(* CODESYS project xlh_rover_signal_test_00_01.project
   Description: Receives some incoming messages and echoes them with CAN-ID +1
   Company: 3S - Smart Software Solutions GmbH
   Version: 1.0.0.0
   Title: CAN Bus API Example
   Author: 3S - Smart Software Solutions GmbH

Project tree, tasks and I/O mapping:
  xLH_base : CODESYS Control for Raspberry Pi 64 SL, CODESYS, order no. 2302000009, version 4.18.0.0
    application app
      libraries: Standard, 3.5.18.0 (System); Util, 3.5.21.0 (System); VisuDialogs, * (System); Memory, * (3S - Smart Software Solutions GmbH); CmpBitmapPool, * (System); CAN API, 1.0.0.4 (CODESYS); MemoryUtils, * (3S - Smart Software Solutions GmbH); CAA CiA 405, 4.3.0.0 (CODESYS)
      task VISU_TASK (cyclic, interval 100 ms, priority 31) calls VisuElems.Visu_Prg
      task MAIN_TASK (cyclic, interval 10 ms, priority 1) calls MAIN_CALLER
      task ENIPAdapterIOTask (cyclic, interval t#1ms, priority 1) calls EtherNet_IP_Adapter.IOCycle
      task ENIPAdapterServiceTask (cyclic, interval t#20ms, priority 30) calls EtherNet_IP_Adapter.ServiceCycle
      program MAIN [ST]
      visualisation Visualization
      program MAIN_CALLER [ST]
      trace Trace (task MAIN_TASK): MAIN.diPosition, MAIN.auiUltrasonic[1], MAIN.iSpeedRight, MAIN.iSpeedLeft, MAIN.iPitch
    SoftMotion General Axis Pool
      a_axis : SM_Drive_PosControl, CODESYS, order no. 1805, version 4.18.0.0
          settings: wDriveID = 4; dwRatioTechUnitsDenom = 101846; iRatioTechUnitsNum = -125; eRampType = 1; fSWMaxVelocity = 50; fSWMaxAcceleration = 100; fSWMaxDeceleration = 100; fSWMaxJerk = 1000; fSWLimitNegative = -1000.0; ScalingIncs = 814768; ScalingUnits = 1000; InvertDirection = TRUE; IsLinearMotor = TRUE; MaximumOutputVelocityInt = 40738; MinimumOutputVelocityInt = -40738; Kp = 0.05; MaxFollowingError = 5.0; EnableFollowingErrorCheck = TRUE; DeadTime = 3.0
      x_axis : SM_Drive_PosControl, CODESYS, order no. 1805, version 4.18.0.0
          settings: dwRatioTechUnitsDenom = 101846; iRatioTechUnitsNum = 125; eRampType = 1; fSWMaxVelocity = 50; fSWMaxAcceleration = 100; fSWMaxDeceleration = 100; fSWMaxJerk = 1000; fSWLimitNegative = -1000; ScalingIncs = 814768; ScalingUnits = 1000; IsLinearMotor = TRUE; MaximumOutputVelocityInt = 40738; MinimumOutputVelocityInt = -40738; Kp = 0.05; MaxFollowingError = 5.0; EnableFollowingErrorCheck = TRUE; DeadTime = 3.0
      y_axis : SM_Drive_PosControl, CODESYS, order no. 1805, version 4.18.0.0
          settings: wDriveID = 2; dwRatioTechUnitsDenom = 101846; iRatioTechUnitsNum = 125; eRampType = 1; fSWMaxVelocity = 50; fSWMaxAcceleration = 100; fSWMaxDeceleration = 100; fSWMaxJerk = 1000; fSWLimitNegative = -1000; ScalingIncs = 814768; ScalingUnits = 1000; IsLinearMotor = TRUE; MaximumOutputVelocityInt = 40738; MinimumOutputVelocityInt = -40738; Kp = 0.05; MaxFollowingError = 5.0; EnableFollowingErrorCheck = TRUE; DeadTime = 3.0
      z_axis : SM_Drive_PosControl, CODESYS, order no. 1805, version 4.18.0.0
          settings: wDriveID = 3; dwRatioTechUnitsDenom = 101846; iRatioTechUnitsNum = 125; eRampType = 1; fSWMaxVelocity = 50; fSWMaxAcceleration = 100; fSWMaxDeceleration = 100; fSWMaxJerk = 1000; fSWLimitNegative = -1000; ScalingIncs = 814768; ScalingUnits = 1000; IsLinearMotor = TRUE; MaximumOutputVelocityInt = 40738; MinimumOutputVelocityInt = -40738; Kp = 0.05; MaxFollowingError = 5.0; EnableFollowingErrorCheck = TRUE; DeadTime = 3.0
    GPIOs_A_B : GPIOs B+/Pi2, CODESYS, version 4.15.0.0
        unmapped channels: digital inputs (GPIO0..GPIO31), digital outputs (GPIO0..GPIO31)
    Onewire
    Camera device
      <Leer>
    SPI
    I²C
    CANbus : CANbus, CODESYS, version 4.3.0.0
        settings: Baudrate = 1000 kbit/s
      CANopen_Manager : CANopen_Manager, CODESYS, version 4.3.0.0
          settings: ConfigVersion = 50659584
        xlh_ddsm210_ultrasonic : xlh_ddsm210_ultrasonic, xemax ag, order no. 0, version Revision=16#00000001, FileVersion=1.0
            settings: NODEIDSAVED = 1; SDO Timeout = 1000000; PDO_Autoconfig = FALSE; EXPERTSETTINGS = FALSE; Sync-General Parameters.Sync-COBID = 16#00000080; Sync-General Parameters.Communication Cycle Period = 16#00000000 usec; PDO 16#1400.COBID = 16#00000201; Process by CANopenManager = TRUE; PDO 16#1800.COBID = 16#00000181; Process by CANopenManager = TRUE; PDO 16#1801.COBID = 16#00000281; Process by CANopenManager = TRUE; PDO 16#1802.COBID = 16#00000381; Process by CANopenManager = TRUE; PDO 16#1803.COBID = 16#00000481; Process by CANopenManager = TRUE; set_speed.Subindex = 16#01; set_current_limit.Subindex = 16#01; set_acc_time.Subindex = 16#01; set_cmd.Subindex = 16#01; speed.Subindex = 16#01; current.Subindex = 16#01; acc_time.Subindex = 16#01; temperature.Subindex = 16#01; position.Subindex = 16#01; error_code.Subindex = 16#01; ultrasonic_1.Subindex = 16#01; ultrasonic_2.Subindex = 16#02; ultrasonic_3.Subindex = 16#03; debug_1.Subindex = 16#02; ultrasonic_4.Subindex = 16#04; ultrasonic_5.Subindex = 16#05; ultrasonic_6.Subindex = 16#06; debug_2.Subindex = 16#03; SDO List.Set COB-ID sync.Index = 16#1005; SDO List.Set COB-ID sync.Subindex = 16#00; SDO List.Set COB-ID sync.Value = 16#00000080; SDO List.Set COB-ID sync.Size = 32; SDO List.Set COB-ID sync.AbortIfError = FALSE; SDO List.Set COB-ID sync.JumpToLine = FALSE;
              SDO List.Set COB-ID sync.Line = 0; SDO List.Set communication cycle period.Index = 16#1006; SDO List.Set communication cycle period.Subindex = 16#00; SDO List.Set communication cycle period.Value = 16#00000000; SDO List.Set communication cycle period.Size = 32; SDO List.Set communication cycle period.AbortIfError = FALSE; SDO List.Set communication cycle period.JumpToLine = FALSE; SDO List.Set communication cycle period.Line = 0; SDO List.Set Guardtime.Index = 16#100C; SDO List.Set Guardtime.Subindex = 16#00; SDO List.Set Guardtime.Value = 16#000000C8; SDO List.Set Guardtime.Size = 16; SDO List.Set Guardtime.AbortIfError = FALSE; SDO List.Set Guardtime.JumpToLine = FALSE; SDO List.Set Guardtime.Line = 0; SDO List.Set Lifetime.Index = 16#100D; SDO List.Set Lifetime.Subindex = 16#00; SDO List.Set Lifetime.Value = 16#00000003; SDO List.Set Lifetime.Size = 8; SDO List.Set Lifetime.AbortIfError = FALSE; SDO List.Set Lifetime.JumpToLine = FALSE; SDO List.Set Lifetime.Line = 0; SDO List.Set Heartbeat Consumer.Index = 16#1016; SDO List.Set Heartbeat Consumer.Subindex = 16#01; SDO List.Set Heartbeat Consumer.Value = 0; SDO List.Set Heartbeat Consumer.Size = 32; SDO List.Set Heartbeat Consumer.AbortIfError = FALSE; SDO List.Set Heartbeat Consumer.JumpToLine = FALSE; SDO List.Set Heartbeat Consumer.Line = 0; SDO List.Disable PDO.Index = 16#1400; SDO List.Disable PDO.Subindex = 16#01; SDO List.Disable PDO.Value = 16#80000201; SDO List.Disable PDO.Size = 32; SDO List.Disable PDO.AbortIfError = FALSE; SDO List.Disable PDO.JumpToLine = FALSE; SDO List.Disable PDO.Line = 0; SDO List.Set transmission type.Index = 16#1400; SDO List.Set transmission type.Subindex = 16#02; SDO List.Set transmission type.Value = 16#FF; SDO List.Set transmission type.Size = 8;
              SDO List.Set transmission type.AbortIfError = FALSE; SDO List.Set transmission type.JumpToLine = FALSE; SDO List.Set transmission type.Line = 0; SDO List.Set and enable COB-ID.Index = 16#1400; SDO List.Set and enable COB-ID.Subindex = 16#01; SDO List.Set and enable COB-ID.Value = 16#00000201; SDO List.Set and enable COB-ID.Size = 32; SDO List.Set and enable COB-ID.AbortIfError = FALSE; SDO List.Set and enable COB-ID.JumpToLine = FALSE; SDO List.Set and enable COB-ID.Line = 0; SDO List.Disable PDO.Index = 16#1800; SDO List.Disable PDO.Subindex = 16#01; SDO List.Disable PDO.Value = 16#80000181; SDO List.Disable PDO.Size = 32; SDO List.Disable PDO.AbortIfError = FALSE; SDO List.Disable PDO.JumpToLine = FALSE; SDO List.Disable PDO.Line = 0; SDO List.Set transmission type.Index = 16#1800; SDO List.Set transmission type.Subindex = 16#02; SDO List.Set transmission type.Value = 16#FF; SDO List.Set transmission type.Size = 8; SDO List.Set transmission type.AbortIfError = FALSE; SDO List.Set transmission type.JumpToLine = FALSE; SDO List.Set transmission type.Line = 0; SDO List.Set inhibit time.Index = 16#1800; SDO List.Set inhibit time.Subindex = 16#03; SDO List.Set inhibit time.Value = 16#0000; SDO List.Set inhibit time.Size = 16; SDO List.Set inhibit time.AbortIfError = FALSE; SDO List.Set inhibit time.JumpToLine = FALSE; SDO List.Set inhibit time.Line = 0; SDO List.Set event time.Index = 16#1800; SDO List.Set event time.Subindex = 16#05; SDO List.Set event time.Value = 16#0000; SDO List.Set event time.Size = 16; SDO List.Set event time.AbortIfError = FALSE; SDO List.Set event time.JumpToLine = FALSE; SDO List.Set event time.Line = 0; SDO List.Set and enable COB-ID.Index = 16#1800; SDO List.Set and enable COB-ID.Subindex = 16#01;
              SDO List.Set and enable COB-ID.Value = 16#00000181; SDO List.Set and enable COB-ID.Size = 32; SDO List.Set and enable COB-ID.AbortIfError = FALSE; SDO List.Set and enable COB-ID.JumpToLine = FALSE; SDO List.Set and enable COB-ID.Line = 0; SDO List.Disable PDO.Index = 16#1801; SDO List.Disable PDO.Subindex = 16#01; SDO List.Disable PDO.Value = 16#80000281; SDO List.Disable PDO.Size = 32; SDO List.Disable PDO.AbortIfError = FALSE; SDO List.Disable PDO.JumpToLine = FALSE; SDO List.Disable PDO.Line = 0; SDO List.Set transmission type.Index = 16#1801; SDO List.Set transmission type.Subindex = 16#02; SDO List.Set transmission type.Value = 16#FF; SDO List.Set transmission type.Size = 8; SDO List.Set transmission type.AbortIfError = FALSE; SDO List.Set transmission type.JumpToLine = FALSE; SDO List.Set transmission type.Line = 0; SDO List.Set inhibit time.Index = 16#1801; SDO List.Set inhibit time.Subindex = 16#03; SDO List.Set inhibit time.Value = 16#0000; SDO List.Set inhibit time.Size = 16; SDO List.Set inhibit time.AbortIfError = FALSE; SDO List.Set inhibit time.JumpToLine = FALSE; SDO List.Set inhibit time.Line = 0; SDO List.Set event time.Index = 16#1801; SDO List.Set event time.Subindex = 16#05; SDO List.Set event time.Value = 16#0000; SDO List.Set event time.Size = 16; SDO List.Set event time.AbortIfError = FALSE; SDO List.Set event time.JumpToLine = FALSE; SDO List.Set event time.Line = 0; SDO List.Set and enable COB-ID.Index = 16#1801; SDO List.Set and enable COB-ID.Subindex = 16#01; SDO List.Set and enable COB-ID.Value = 16#00000281; SDO List.Set and enable COB-ID.Size = 32; SDO List.Set and enable COB-ID.AbortIfError = FALSE; SDO List.Set and enable COB-ID.JumpToLine = FALSE; SDO List.Set and enable COB-ID.Line = 0;
              SDO List.Disable PDO.Index = 16#1802; SDO List.Disable PDO.Subindex = 16#01; SDO List.Disable PDO.Value = 16#80000381; SDO List.Disable PDO.Size = 32; SDO List.Disable PDO.AbortIfError = FALSE; SDO List.Disable PDO.JumpToLine = FALSE; SDO List.Disable PDO.Line = 0; SDO List.Set transmission type.Index = 16#1802; SDO List.Set transmission type.Subindex = 16#02; SDO List.Set transmission type.Value = 16#FF; SDO List.Set transmission type.Size = 8; SDO List.Set transmission type.AbortIfError = FALSE; SDO List.Set transmission type.JumpToLine = FALSE; SDO List.Set transmission type.Line = 0; SDO List.Set inhibit time.Index = 16#1802; SDO List.Set inhibit time.Subindex = 16#03; SDO List.Set inhibit time.Value = 16#0000; SDO List.Set inhibit time.Size = 16; SDO List.Set inhibit time.AbortIfError = FALSE; SDO List.Set inhibit time.JumpToLine = FALSE; SDO List.Set inhibit time.Line = 0; SDO List.Set event time.Index = 16#1802; SDO List.Set event time.Subindex = 16#05; SDO List.Set event time.Value = 16#0000; SDO List.Set event time.Size = 16; SDO List.Set event time.AbortIfError = FALSE; SDO List.Set event time.JumpToLine = FALSE; SDO List.Set event time.Line = 0; SDO List.Set and enable COB-ID.Index = 16#1802; SDO List.Set and enable COB-ID.Subindex = 16#01; SDO List.Set and enable COB-ID.Value = 16#00000381; SDO List.Set and enable COB-ID.Size = 32; SDO List.Set and enable COB-ID.AbortIfError = FALSE; SDO List.Set and enable COB-ID.JumpToLine = FALSE; SDO List.Set and enable COB-ID.Line = 0; SDO List.Disable PDO.Index = 16#1803; SDO List.Disable PDO.Subindex = 16#01; SDO List.Disable PDO.Value = 16#80000481; SDO List.Disable PDO.Size = 32; SDO List.Disable PDO.AbortIfError = FALSE;
              SDO List.Disable PDO.JumpToLine = FALSE; SDO List.Disable PDO.Line = 0; SDO List.Set transmission type.Index = 16#1803; SDO List.Set transmission type.Subindex = 16#02; SDO List.Set transmission type.Value = 16#FF; SDO List.Set transmission type.Size = 8; SDO List.Set transmission type.AbortIfError = FALSE; SDO List.Set transmission type.JumpToLine = FALSE; SDO List.Set transmission type.Line = 0; SDO List.Set inhibit time.Index = 16#1803; SDO List.Set inhibit time.Subindex = 16#03; SDO List.Set inhibit time.Value = 16#0000; SDO List.Set inhibit time.Size = 16; SDO List.Set inhibit time.AbortIfError = FALSE; SDO List.Set inhibit time.JumpToLine = FALSE; SDO List.Set inhibit time.Line = 0; SDO List.Set event time.Index = 16#1803; SDO List.Set event time.Subindex = 16#05; SDO List.Set event time.Value = 16#0000; SDO List.Set event time.Size = 16; SDO List.Set event time.AbortIfError = FALSE; SDO List.Set event time.JumpToLine = FALSE; SDO List.Set event time.Line = 0; SDO List.Set and enable COB-ID.Index = 16#1803; SDO List.Set and enable COB-ID.Subindex = 16#01; SDO List.Set and enable COB-ID.Value = 16#00000481; SDO List.Set and enable COB-ID.Size = 32; SDO List.Set and enable COB-ID.AbortIfError = FALSE; SDO List.Set and enable COB-ID.JumpToLine = FALSE; SDO List.Set and enable COB-ID.Line = 0; ConfigVersion = 50659584
            output app.MAIN.iSetSpeedLeft : INT  // set_speed
            output app.MAIN.iSetCurrentLimit : INT  // set_current_limit
            output app.MAIN.bySetAccTime : USINT  // set_acc_time
            output app.MAIN.bySetCmd : USINT  // set_cmd
            input  app.MAIN.iSpeedLeft : INT  // speed
            input  app.MAIN.iCurrentLeft : INT  // current
            input  app.MAIN.byAccTimeLeft : USINT  // acc_time
            input  app.MAIN.byTemperatureLeft : USINT  // temperature
            input  app.MAIN.diPositionLeft : DINT  // position
            input  app.MAIN.uiErrorCodeLeft : UINT  // error_code
            input  app.MAIN.uiUltrasonicRear : UINT  // ultrasonic_1
            input  app.MAIN.uiUltrasonicRearRight : UINT  // ultrasonic_2
            input  app.MAIN.uiUltrasonicFrontRight : UINT  // ultrasonic_3
            input  app.MAIN.uiUltrasonicFront : UINT  // ultrasonic_4
            input  app.MAIN.uiUltrasonicFrontLeft : UINT  // ultrasonic_5
            input  app.MAIN.uiUltrasonicRearLeft : UINT  // ultrasonic_6
            unmapped channels: debug_1, debug_2
        xlh_ddsm210_imu : xlh_ddsm210_imu, xemax ag, order no. 0, version Revision=16#00000001, FileVersion=1.0
            settings: NODEIDSAVED = 2; SDO Timeout = 1000000; EXPERTSETTINGS = FALSE; Sync-General Parameters.Sync-COBID = 16#00000080; Sync-General Parameters.Communication Cycle Period = 16#00000000 usec; PDO 16#1400.COBID = 16#00000202; Process by CANopenManager = TRUE; PDO 16#1800.COBID = 16#00000182; Process by CANopenManager = TRUE; PDO 16#1801.COBID = 16#00000282; Process by CANopenManager = TRUE; PDO 16#1802.COBID = 16#00000382; Process by CANopenManager = TRUE; set_speed.Subindex = 16#01; set_current_limit.Subindex = 16#01; set_acc_time.Subindex = 16#01; set_cmd.Subindex = 16#01; speed.Subindex = 16#01; current.Subindex = 16#01; acc_time.Subindex = 16#01; temperature.Subindex = 16#01; position.Subindex = 16#01; error_code.Subindex = 16#01; debug_1.Subindex = 16#02; yaw.Subindex = 16#01; pitch.Subindex = 16#02; roll.Subindex = 16#03; debug_2.Subindex = 16#03; SDO List.Set COB-ID sync.Index = 16#1005; SDO List.Set COB-ID sync.Subindex = 16#00; SDO List.Set COB-ID sync.Value = 16#00000080; SDO List.Set COB-ID sync.Size = 32; SDO List.Set COB-ID sync.AbortIfError = FALSE; SDO List.Set COB-ID sync.JumpToLine = FALSE; SDO List.Set COB-ID sync.Line = 0; SDO List.Set communication cycle period.Index = 16#1006; SDO List.Set communication cycle period.Subindex = 16#00; SDO List.Set communication cycle period.Value = 16#00000000; SDO List.Set communication cycle period.Size = 32; SDO List.Set communication cycle period.AbortIfError = FALSE;
              SDO List.Set communication cycle period.JumpToLine = FALSE; SDO List.Set communication cycle period.Line = 0; SDO List.Set Guardtime.Index = 16#100C; SDO List.Set Guardtime.Subindex = 16#00; SDO List.Set Guardtime.Value = 16#000000C8; SDO List.Set Guardtime.Size = 16; SDO List.Set Guardtime.AbortIfError = FALSE; SDO List.Set Guardtime.JumpToLine = FALSE; SDO List.Set Guardtime.Line = 0; SDO List.Set Lifetime.Index = 16#100D; SDO List.Set Lifetime.Subindex = 16#00; SDO List.Set Lifetime.Value = 16#00000003; SDO List.Set Lifetime.Size = 8; SDO List.Set Lifetime.AbortIfError = FALSE; SDO List.Set Lifetime.JumpToLine = FALSE; SDO List.Set Lifetime.Line = 0; SDO List.Set Heartbeat Consumer.Index = 16#1016; SDO List.Set Heartbeat Consumer.Subindex = 16#01; SDO List.Set Heartbeat Consumer.Value = 0; SDO List.Set Heartbeat Consumer.Size = 32; SDO List.Set Heartbeat Consumer.AbortIfError = FALSE; SDO List.Set Heartbeat Consumer.JumpToLine = FALSE; SDO List.Set Heartbeat Consumer.Line = 0; SDO List.Disable PDO.Index = 16#1400; SDO List.Disable PDO.Subindex = 16#01; SDO List.Disable PDO.Value = 16#80000202; SDO List.Disable PDO.Size = 32; SDO List.Disable PDO.AbortIfError = FALSE; SDO List.Disable PDO.JumpToLine = FALSE; SDO List.Disable PDO.Line = 0; SDO List.Set transmission type.Index = 16#1400; SDO List.Set transmission type.Subindex = 16#02; SDO List.Set transmission type.Value = 16#FF; SDO List.Set transmission type.Size = 8; SDO List.Set transmission type.AbortIfError = FALSE; SDO List.Set transmission type.JumpToLine = FALSE; SDO List.Set transmission type.Line = 0; SDO List.Set and enable COB-ID.Index = 16#1400; SDO List.Set and enable COB-ID.Subindex = 16#01; SDO List.Set and enable COB-ID.Value = 16#00000202;
              SDO List.Set and enable COB-ID.Size = 32; SDO List.Set and enable COB-ID.AbortIfError = FALSE; SDO List.Set and enable COB-ID.JumpToLine = FALSE; SDO List.Set and enable COB-ID.Line = 0; SDO List.Disable PDO.Index = 16#1800; SDO List.Disable PDO.Subindex = 16#01; SDO List.Disable PDO.Value = 16#80000182; SDO List.Disable PDO.Size = 32; SDO List.Disable PDO.AbortIfError = FALSE; SDO List.Disable PDO.JumpToLine = FALSE; SDO List.Disable PDO.Line = 0; SDO List.Set transmission type.Index = 16#1800; SDO List.Set transmission type.Subindex = 16#02; SDO List.Set transmission type.Value = 16#FF; SDO List.Set transmission type.Size = 8; SDO List.Set transmission type.AbortIfError = FALSE; SDO List.Set transmission type.JumpToLine = FALSE; SDO List.Set transmission type.Line = 0; SDO List.Set inhibit time.Index = 16#1800; SDO List.Set inhibit time.Subindex = 16#03; SDO List.Set inhibit time.Value = 16#0000; SDO List.Set inhibit time.Size = 16; SDO List.Set inhibit time.AbortIfError = FALSE; SDO List.Set inhibit time.JumpToLine = FALSE; SDO List.Set inhibit time.Line = 0; SDO List.Set event time.Index = 16#1800; SDO List.Set event time.Subindex = 16#05; SDO List.Set event time.Value = 16#0000; SDO List.Set event time.Size = 16; SDO List.Set event time.AbortIfError = FALSE; SDO List.Set event time.JumpToLine = FALSE; SDO List.Set event time.Line = 0; SDO List.Set and enable COB-ID.Index = 16#1800; SDO List.Set and enable COB-ID.Subindex = 16#01; SDO List.Set and enable COB-ID.Value = 16#00000182; SDO List.Set and enable COB-ID.Size = 32; SDO List.Set and enable COB-ID.AbortIfError = FALSE; SDO List.Set and enable COB-ID.JumpToLine = FALSE; SDO List.Set and enable COB-ID.Line = 0; SDO List.Disable PDO.Index = 16#1801;
              SDO List.Disable PDO.Subindex = 16#01; SDO List.Disable PDO.Value = 16#80000282; SDO List.Disable PDO.Size = 32; SDO List.Disable PDO.AbortIfError = FALSE; SDO List.Disable PDO.JumpToLine = FALSE; SDO List.Disable PDO.Line = 0; SDO List.Set transmission type.Index = 16#1801; SDO List.Set transmission type.Subindex = 16#02; SDO List.Set transmission type.Value = 16#FF; SDO List.Set transmission type.Size = 8; SDO List.Set transmission type.AbortIfError = FALSE; SDO List.Set transmission type.JumpToLine = FALSE; SDO List.Set transmission type.Line = 0; SDO List.Set inhibit time.Index = 16#1801; SDO List.Set inhibit time.Subindex = 16#03; SDO List.Set inhibit time.Value = 16#0000; SDO List.Set inhibit time.Size = 16; SDO List.Set inhibit time.AbortIfError = FALSE; SDO List.Set inhibit time.JumpToLine = FALSE; SDO List.Set inhibit time.Line = 0; SDO List.Set event time.Index = 16#1801; SDO List.Set event time.Subindex = 16#05; SDO List.Set event time.Value = 16#0000; SDO List.Set event time.Size = 16; SDO List.Set event time.AbortIfError = FALSE; SDO List.Set event time.JumpToLine = FALSE; SDO List.Set event time.Line = 0; SDO List.Set and enable COB-ID.Index = 16#1801; SDO List.Set and enable COB-ID.Subindex = 16#01; SDO List.Set and enable COB-ID.Value = 16#00000282; SDO List.Set and enable COB-ID.Size = 32; SDO List.Set and enable COB-ID.AbortIfError = FALSE; SDO List.Set and enable COB-ID.JumpToLine = FALSE; SDO List.Set and enable COB-ID.Line = 0; SDO List.Disable PDO.Index = 16#1802; SDO List.Disable PDO.Subindex = 16#01; SDO List.Disable PDO.Value = 16#80000382; SDO List.Disable PDO.Size = 32; SDO List.Disable PDO.AbortIfError = FALSE; SDO List.Disable PDO.JumpToLine = FALSE;
              SDO List.Disable PDO.Line = 0; SDO List.Set transmission type.Index = 16#1802; SDO List.Set transmission type.Subindex = 16#02; SDO List.Set transmission type.Value = 16#FF; SDO List.Set transmission type.Size = 8; SDO List.Set transmission type.AbortIfError = FALSE; SDO List.Set transmission type.JumpToLine = FALSE; SDO List.Set transmission type.Line = 0; SDO List.Set inhibit time.Index = 16#1802; SDO List.Set inhibit time.Subindex = 16#03; SDO List.Set inhibit time.Value = 16#0000; SDO List.Set inhibit time.Size = 16; SDO List.Set inhibit time.AbortIfError = FALSE; SDO List.Set inhibit time.JumpToLine = FALSE; SDO List.Set inhibit time.Line = 0; SDO List.Set event time.Index = 16#1802; SDO List.Set event time.Subindex = 16#05; SDO List.Set event time.Value = 16#0000; SDO List.Set event time.Size = 16; SDO List.Set event time.AbortIfError = FALSE; SDO List.Set event time.JumpToLine = FALSE; SDO List.Set event time.Line = 0; SDO List.Set and enable COB-ID.Index = 16#1802; SDO List.Set and enable COB-ID.Subindex = 16#01; SDO List.Set and enable COB-ID.Value = 16#00000382; SDO List.Set and enable COB-ID.Size = 32; SDO List.Set and enable COB-ID.AbortIfError = FALSE; SDO List.Set and enable COB-ID.JumpToLine = FALSE; SDO List.Set and enable COB-ID.Line = 0; ConfigVersion = 50659584
            output app.MAIN.iSetSpeedRight : INT  // set_speed
            output app.MAIN.iSetCurrentLimit : INT  // set_current_limit
            output app.MAIN.bySetAccTime : USINT  // set_acc_time
            output app.MAIN.bySetCmd : USINT  // set_cmd
            input  app.MAIN.iSpeedRight : INT  // speed
            input  app.MAIN.iCurrentRight : INT  // current
            input  app.MAIN.byAccTimeRight : USINT  // acc_time
            input  app.MAIN.byTemperatureRight : USINT  // temperature
            input  app.MAIN.diPositionRight : DINT  // position
            input  app.MAIN.uiErrorCodeRight : UINT  // error_code
            input  app.MAIN.iYaw : INT  // yaw
            input  app.MAIN.iPitch : INT  // pitch
            input  app.MAIN.iRoll : INT  // roll
            unmapped channels: debug_1, debug_2
    Ethernet : Ethernet, CODESYS, version 4.2.0.0
        settings: IPAddress = [192,168,1,189]; SubnetMask = [255,255,255,0]; GatewayAddress = [192,168,1,1]; MACAddress = [16#00,16#00,16#00,16#00,16#00,16#00]; NetworkInterfaceName = 'wlan0'; NetworkInterfaceName = "wlan0"; SaveCommunicationSettings = FALSE; IPAddress = [192,168,0,2]; SubnetMask = [255,255,255,0]; GatewayAddress = [0,0,0,0]
      EtherNet_IP_Adapter : EtherNet/IP Adapter, CODESYS, version 4.8.0.0
          settings: DeviceInfo.ProductName = 'xlh_rover_signal_test'; DeviceInfo.ProductCode = 1101; DeviceInfo.MajorRevision = 2; Number of Assemblies = 5; Number of Connections = 3; Connection Settings.Connection Number = 0; Connection Settings.Trigger and Transport = 67305474; Connection Settings.Connection Parameters = 4284744709; Connection Settings.O->T Requested packet interval (µs) = 0; Connection Settings.O->T Size (Bytes) = 0; Connection Settings.T->O Requested packet interval (µs) = 0; Connection Settings.T->O Size (Bytes) = 0; Connection Settings.Target Config Size (Bytes) = 2; Connection Settings.Connection Path Size (Bytes) = 8; Connection Settings.Connection Number = 1; Connection Settings.Trigger and Transport = 33751042; Connection Settings.Connection Parameters = 4284744453; Connection Settings.O->T Requested packet interval (µs) = 0; Connection Settings.O->T Size (Bytes) = 0; Connection Settings.T->O Requested packet interval (µs) = 0; Connection Settings.T->O Size (Bytes) = 0; Connection Settings.Target Config Size (Bytes) = 0; Connection Settings.Connection Path Size (Bytes) = 6; Connection Settings.Connection Number = 2; Connection Settings.Trigger and Transport = 16973826; Connection Settings.Connection Parameters = 4284744453; Connection Settings.O->T Requested packet interval (µs) = 0; Connection Settings.O->T Size (Bytes) = 0; Connection Settings.T->O Requested packet interval (µs) = 0; Connection Settings.T->O Size (Bytes) = 0; Connection Settings.Target Config Size (Bytes) = 0; Connection Settings.Connection Path Size (Bytes) = 6; Connection Path = [16#20,16#04,16#24,16#66,16#2C,16#64,16#2C,16#65]; Connection Path = [16#20,16#04,16#2C,16#C6,16#2C,16#65]; Connection Path = [16#20,16#04,16#2C,16#C7,16#2C,16#65]; Default Connection Path = [16#20,16#04,16#24,16#66,16#2C,16#64,16#2C,16#65]; Default Connection Path = [16#20,16#04,16#2C,16#C6,16#2C,16#65]; Default Connection Path = [16#20,16#04,16#2C,16#C7,16#2C,16#65]
        EtherNet_IP_Module : EtherNet/IP Module, CODESYS, version 4.6.0.0
            settings: ConsumingAssemblyID = 100; ProducingAssemblyID = 101; fJoystickXnorm.ReadOnly = False; fJoystickXnorm.BitSize = 64; fJoystickXnorm.DataSize = 8; fJoystickYnorm.ReadOnly = False; fJoystickYnorm.BitSize = 64; fJoystickYnorm.DataSize = 8; bySwitch.ReadOnly = False; byButton.ReadOnly = False; byLedSwitch.ReadOnly = False; byLedButton.ReadOnly = False; ConfigVersion = 50663168
            input  app.MAIN.fJoystickXnorm : LREAL  // fJoystickXnorm
            input  app.MAIN.fJoystickYnorm : LREAL  // fJoystickYnorm
            input  app.MAIN.bySwitch : BYTE  // bySwitch
            input  app.MAIN.byButton : BYTE  // byButton
            output app.MAIN.byLedSwitch : BYTE  // byLedSwitch
            output app.MAIN.byLedButton : BYTE  // byLedButton
  libraries: VisuSymbols, 4.5.0.0 (System); DepictorBase, 1.2.0.0 (CODESYS)
  text list GlobalTextList
  5ce3da45-db07-42e7-a21c-a00fff4ed8f6|C:\Users\phe\Downloads\Musterloesung_FUP.PNG
*)

// xLH_base/app/MAIN_CALLER
PROGRAM MAIN_CALLER
VAR
	bDevicesCoRunning: BOOL;
	fbTonDevicesCoRunning: TON := (PT:=T#250MS);
END_VAR

// Ueberwachung ob alle CAN-Open Devices im Status RUN sind
fbTonDevicesCoRunning(IN:= 
	(xlh_ddsm210_ultrasonic.CANopenState = _3SCOS.DEVICE_STATE.OPERATIONAL) AND
	(xlh_ddsm210_imu.CANopenState = _3SCOS.DEVICE_STATE.OPERATIONAL)
);

// falls alle Devices im Status RUN sind (inklusive Verzögerung), wird die POE MAIN aufgerufen
IF fbTonDevicesCoRunning.Q THEN
	MAIN();
END_IF

END_PROGRAM

// xLH_base/app/MAIN
PROGRAM MAIN
VAR_INPUT
	iSpeedLeft: INT;
	iSpeedRight: INT;
	iCurrentLeft: INT;
	iCurrentRight: INT;
	byAccTimeLeft: BYTE;
	byAccTimeRight: BYTE;
	byTemperatureLeft: BYTE;
	byTemperatureRight: BYTE;
	diPositionLeft: DINT;// still errors in the calculation => set to zero in the fw
	diPositionRight: DINT;// still errors in the calculation => set to zero in the fw
	{attribute 'displaymode':='hex'} 
	uiErrorCodeLeft: UINT;
	uiErrorCodeRight: UINT;
	uiUltrasonicFront: UINT;
	uiUltrasonicFrontLeft: UINT;
	uiUltrasonicFrontRight: UINT;
	uiUltrasonicRear: UINT;
	uiUltrasonicRearLeft: UINT;
	uiUltrasonicRearRight: UINT;
	
	
	iYaw: INT;
	iPitch: INT;
	iRoll: INT;
	fYaw: LREAL;
	fPitch: LREAL;
	fRoll: LREAL;
	
	// Ethernet IP
	fJoystickXnorm: LREAL;
	fJoystickYnorm: LREAL;
	bySwitch: BYTE;
	byButton: BYTE;
	iDebugRead: INT;
END_VAR
VAR_OUTPUT
	iSetSpeedLeft: INT := 0;
	iSetSpeedRight: INT := 0;
	iSetCurrentLimit: INT := 1000;// deactivated in the fw
	bySetAccTime: BYTE := 5;
	bySetCmd: BYTE := 0;
	
	// Ethernet IP
	byLedSwitch: BYTE;
	byLedButton: BYTE;
	iDebugWrite: INT;
END_VAR
VAR
	fSetSpeedLeft: LREAL;
	fSetSpeedRight: LREAL;
	
	byDummy: BYTE;
	iDummy: INT;
	uiDummy: UINT;
	diDummy: DINT;
	udiDummy: UDINT;

	fbBlink: BLINK := (TIMEHIGH:=T#100MS, TIMELOW:=T#100MS, ENABLE:=TRUE);
	fDummy: LREAL;
	
	unpackByte: MEM.UnpackByte;	
	abSwitch: ARRAY [0..7] OF BOOL;
	abButton: ARRAY [0..7] OF BOOL;
END_VAR
VAR CONSTANT
	fSpeedMax: LREAL := 500.0;
	fSpeedMaxDir: LREAL := 250.0;
END_VAR

fSetSpeedLeft := fJoystickYnorm * fSpeedMax * (1.0) + ABS(MAX(fJoystickXnorm, 0.0)) * fSpeedMaxDir * (1.0);
fSetSpeedRight := fJoystickYnorm * fSpeedMax * (-1.0) + ABS(MIN(fJoystickXnorm, 0.0)) * fSpeedMaxDir * (-1.0);

iSetSpeedLeft := TO_INT(fSetSpeedLeft);
iSetSpeedRight := TO_INT(fSetSpeedRight);
byDummy := bySetAccTime;

iDummy := iSpeedLeft;// -2100 ~ 2100 -> -210 ~ 210 rpm
iDummy := iSpeedRight;// -2100 ~ 2100 -> -210 ~ 210 rpm
iDummy := iCurrentLeft;// mA
iDummy := iCurrentRight;// mA
byDummy := byAccTimeLeft;// When it is set to 1, the acceleration time per 1rpm is 0.1ms. When it is set to 10, the acceleration time per 1rpm is 10*0.1 ms=1ms.
byDummy := byTemperatureLeft;// °C
uiDummy := uiUltrasonicFront;// resolution 0.1mm => 1000 ~ 100.0mm
uiDummy := uiUltrasonicFrontRight;// resolution 0.1mm => 1000 ~ 100.0mm
uiDummy := uiUltrasonicFrontLeft;// resolution 0.1mm => 1000 ~ 100.0mm
uiDummy := uiUltrasonicRear;// resolution 0.1mm => 1000 ~ 100.0mm
uiDummy := uiUltrasonicRearRight;// resolution 0.1mm => 1000 ~ 100.0mm
uiDummy := uiUltrasonicRearLeft;// resolution 0.1mm => 1000 ~ 100.0mm
uiDummy := uiErrorCodeLeft;

iDummy := iYaw;// resolution 0.01°
iDummy := iPitch;// resolution 0.01°
iDummy := iRoll;// resolution 0.01°
fYaw := TO_LREAL(iYaw) * 0.01;
fPitch := TO_LREAL(iPitch) * 0.01;
fRoll := TO_LREAL(iRoll) * 0.01; 

// Ethernet IP
fDummy := fJoystickXnorm;
fDummy := fJoystickYnorm;
byDummy := bySwitch;
byDummy := byButton;
iDummy := iDebugRead;

byDummy := byLedSwitch;
byDummy := byLedButton;
iDebugWrite := iDebugRead + 1;// Performancetester

byLedSwitch := MEM.PackBitsToByte(
		FALSE,
		FALSE,
		FALSE,
		FALSE,
		FALSE,
		FALSE,
		FALSE,
		fbBlink.OUT and abSwitch[0]);
		
byLedButton := MEM.PackBitsToByte(
		fbBlink.OUT AND abButton[7],
		FALSE,
		FALSE,
		FALSE,
		FALSE,
		FALSE,
		FALSE,
		FALSE);

unpackByte(byValue := bySwitch);	
abSwitch[0] := unpackByte.xBit0;
abSwitch[1] := unpackByte.xBit1;
abSwitch[2] := unpackByte.xBit2;
abSwitch[3] := unpackByte.xBit3;
abSwitch[4] := unpackByte.xBit4;
abSwitch[5] := unpackByte.xBit5;
abSwitch[6] := unpackByte.xBit6;
abSwitch[7] := unpackByte.xBit7;

unpackByte(byValue := byButton);	
abButton[0] := unpackByte.xBit0;
abButton[1] := unpackByte.xBit1;
abButton[2] := unpackByte.xBit2;
abButton[3] := unpackByte.xBit3;
abButton[4] := unpackByte.xBit4;
abButton[5] := unpackByte.xBit5;
abButton[6] := unpackByte.xBit6;
abButton[7] := unpackByte.xBit7;

END_PROGRAM

// xLH_base/app/Visualization
VISUALIZATION Visualization  // 2x2
END_VISUALIZATION
